(*
SPDX-FileCopyrightText: © 2026 Oleksandr Tiutyk <trofimich@gmail.com>
SPDX-License-Identifier: MIT
License: https://opensource.org/license/mit
*)

{attribute 'qualified_only'}
{attribute 'to_string'}
TYPE EXCEPTION_REACTION :
(
	SET_ERROR_AND_STOP,
	SET_ERROR_AND_CONTINUE,
	IGNORE
);
END_TYPE

(* stored: Version 1.1.0.1
   DUT EXCEPTION_REACTION: Id {774d76d6-0135-4bca-b6fc-6df41659ea71} *)
